FUNCTION_BLOCK FB_SimplePulseGenerator
VAR_INPUT
	IbGenerate	AT%I*	:	BOOL;
	tPulseLength		:	TIME;		
END_VAR
VAR_OUTPUT
	QbOut		AT%Q*	:	BOOL;
END_VAR
VAR
	ton					:	TON;
	rtIn				:	R_TRIG;
	iCase				:	INT;
END_VAR

rtIn		(	CLK		:=	IbGenerate						);
ton			(	IN		:=	QbOut,	PT	:=	tPulseLength	);

IF (NOT QbOut AND rtIn.Q) THEN
	QbOut										:=	TRUE;
ELSIF (ton.Q) THEN
	QbOut										:=	FALSE;	
END_IF

END_FUNCTION_BLOCK

(* stored: Version 1.2.0.0, ProductVersion 3.1.4026.13, FileIdentifier 378b4bd251f8743b949873120dc46a8e13528aaf, FileSignature 78b53edfba15531f67dd4d8b96acb1c1ad4718d7d765075e04395ce1fe630a3fac94410af6472380959f9ebc91b353b4a9b87241f5188900830e2bc8831973e956492440c74c39102d8f77e38fcd9261958af1c255dc153376d6ebebac82fc26db767b263870e3df201e09bb7b771dac19c3fdd9411d6cbc0c744e587e77cecbebaa42f2c291564ce80dc134fe2d329d1677dbee1e71ead8584743247b3fb7852adc7029078735958e8dbd062bba0f14fd9a3277ce9b1186164ca06e8ce064569f12635d294a39221c35a2637b3d9104920aa9d0859b1899755714df9947c827dc8e57c1c94657f6c5a70879de681d08032023903b672fec8459d35a005fd588
   POU FB_SimplePulseGenerator: Id {16cc4e08-d339-44fa-9305-eb23980b6241}, SpecialFunc None *)
